// TIA Portal project "Assembler" (V15)
// Vorlageprojekt für das Buch mit Zielsystem S7-1200

(* hardware
DEVICE "S7-1200-Station_1"  S7-1200 Station
   slot 0: "Baugruppenträger_0"  Rack  V1.0
   slot 1: "PLC_1"  CPU 1211C DC/DC/DC  6ES7 211-1AE40-0XB0  V4.1
*)

// ===== PLC "PLC_1"  CPU 1211C DC/DC/DC =====

VAR_GLOBAL   // PLC tag table "Standard-Variablentabelle"
   "Clock_Byte" AT %MB0 : Byte;
   "Clock_10Hz" AT %M0.0 : Bool;
   "Clock_5Hz" AT %M0.1 : Bool;
   "Clock_2.5Hz" AT %M0.2 : Bool;
   "Clock_2Hz" AT %M0.3 : Bool;
   "Clock_1.25Hz" AT %M0.4 : Bool;
   "Clock_1Hz" AT %M0.5 : Bool;
   "Clock_0.625Hz" AT %M0.6 : Bool;
   "Clock_0.5Hz" AT %M0.7 : Bool;
END_VAR

VAR_GLOBAL   // PLC tag table "Assembler"
   "Moving X" AT %I0.0 : Bool;   // Moving X
   "Moving Z" AT %I0.1 : Bool;   // Moving Z
   "Item detected" AT %I0.2 : Bool;   // Item detected
   "Lid at place" AT %I0.3 : Bool;   // Lid at place
   "Lid clamped" AT %I0.4 : Bool;   // Lid clamped
   "Pos. at limit (lids)" AT %I0.5 : Bool;   // Pos. at limit (lids) (NC)
   "Base at place" AT %I0.6 : Bool;   // Base at place
   "Base clamped" AT %I0.7 : Bool;   // Base clamped
   "Pos. at limit (bases)" AT %I1.0 : Bool;   // Pos. at limit (bases) (NC)
   "Part leaving" AT %I1.1 : Bool;   // Part leaving
   "Start" AT %I1.2 : Bool;   // Start
   "Reset" AT %I1.3 : Bool;   // Reset
   "Stop" AT %I1.4 : Bool;   // Stop (NC)
   "Emergency stop" AT %I1.5 : Bool;   // Emergency stop (NC)
   "Auto" AT %I1.6 : Bool;   // Auto
   "FACTORY I/O (Running)" AT %I1.7 : Bool;   // FACTORY I/O (Running)
   "Move X" AT %Q0.0 : Bool;   // Move X
   "Move Z" AT %Q0.1 : Bool;   // Move Z
   "Grab" AT %Q0.2 : Bool;   // Grab
   "Lids conveyor" AT %Q0.3 : Bool;   // Lids conveyor
   "Clamp lid" AT %Q0.4 : Bool;   // Clamp lid
   "Pos. raise (lids)" AT %Q0.5 : Bool;   // Pos. raise (lids)
   "Bases conveyor" AT %Q0.6 : Bool;   // Bases conveyor
   "Clamp base" AT %Q0.7 : Bool;   // Clamp base
   "Pos. raise (bases)" AT %Q1.0 : Bool;   // Pos. raise (bases)
   "Start light" AT %Q1.1 : Bool;   // Start light
   "Reset light" AT %Q1.2 : Bool;   // Reset light
   "Stop light" AT %Q1.3 : Bool;   // Stop light
   "Counter" AT %QW30 : Int;   // Counter
END_VAR

VAR_GLOBAL   // PLC tag table "GRAFCET"
   "memReset" AT %M2.0 : Bool;   // memReset
   "memStepsOff" AT %M2.1 : Bool;   // memStepsOff
   "memInit" AT %M2.2 : Bool;   // memInit
   "Step 1" AT %M2.3 : Bool;   // Step 1
   "Step 2" AT %M2.4 : Bool;   // Step 2
   "Step 3" AT %M2.5 : Bool;   // Step 3
   "Step 4" AT %M2.6 : Bool;   // Step 4
   "Step 5" AT %M2.7 : Bool;   // Step 5
   "Step 6" AT %M3.0 : Bool;   // Step 6
   "Step 7" AT %M3.1 : Bool;   // Step 7
   "Step 8" AT %M3.2 : Bool;   // Step 8
   "Step 9" AT %M3.3 : Bool;   // Step 9
   "Step 10" AT %M3.4 : Bool;   // Step 10
   "Step 11" AT %M3.5 : Bool;   // Step 11
   "Step 12" AT %M3.6 : Bool;   // Step 12
   "Step 13" AT %M3.7 : Bool;   // Step 13
   "Step 14" AT %M4.0 : Bool;   // Step 14
   "Step 15" AT %M4.1 : Bool;   // Step 15
   "N Lid at place" AT %M4.2 : Bool;   // Neg edge for Lid at place
   "N Base at place" AT %M4.3 : Bool;   // Neg edge for Base at place
   "N Moving Z1" AT %M4.4 : Bool;   // Neg edge for Moving Z1
   "N Moving X" AT %M4.6 : Bool;   // Neg edge for Moving X
   "N Part leaving" AT %M4.7 : Bool;   // Neg edge for Part leaving
   "N Moving Z2" AT %M4.5 : Bool;   // Neg edge for Moving Z2
   "Auto Flag" AT %M5.0 : Bool;   // Auto Flag
   "Manual Flag" AT %M5.1 : Bool;   // Manual Flag
END_VAR

// folder: System blocks/Program resources

DATA_BLOCK "Parts Counter"   // DB1
{ S7_Optimized_Access := 'TRUE' }
AUTHOR : Simatic
FAMILY : IEC
NAME : CNTR
VERSION : 1.0
// stored: InstanceOfName IEC_COUNTER
"IEC_COUNTER"
BEGIN
END_DATA_BLOCK

// folder: (top level)

FUNCTION "Steps" : Void   // FC1, LAD
{ S7_Optimized_Access := 'TRUE' }
VERSION : 0.1
   VAR_TEMP   // added for the SCL form of the ladder/FBD networks
      _w1 : Bool;
   END_VAR
BEGIN

REGION Network 1: Manual Flag
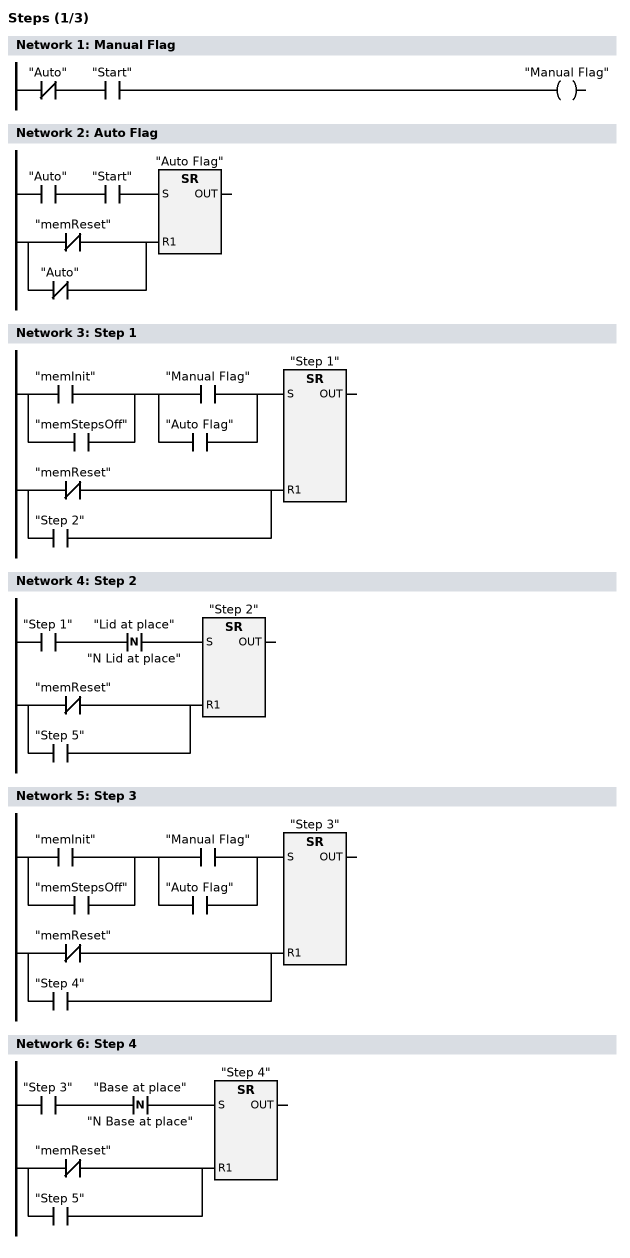
   RUNG wire#powerrail
      I_Contact( "Auto" )
      Contact( "Start" )
      Coil( "Manual Flag" )
   END_RUNG
   // the same network as SCL:
   "Manual Flag" := NOT "Auto" AND "Start";
END_REGION

REGION Network 2: Auto Flag
   RUNG wire#powerrail
      Contact( "Auto" )
      Contact( "Start" )
      S_SR(operand := "Auto Flag", r1 := wire#w1)
   END_RUNG
   RUNG wire#powerrail
      I_Contact( "memReset" )
   END_RUNG wire#w1
   RUNG wire#powerrail
      I_Contact( "Auto" )
   END_RUNG wire#w1
   // the same network as SCL:
   IF "Auto" AND "Start" THEN
       "Auto Flag" := TRUE;   // SR flip-flop
   END_IF;
   IF NOT "memReset" OR NOT "Auto" THEN "Auto Flag" := FALSE; END_IF;
END_REGION

REGION Network 3: Step 1
   RUNG wire#powerrail
      Contact( "memInit" )
      wire#w1
      Contact( "Manual Flag" )
      wire#w2
      S_SR(operand := "Step 1", r1 := wire#w3)
   END_RUNG
   RUNG wire#powerrail
      Contact( "memStepsOff" )
   END_RUNG wire#w1
   RUNG wire#w1
      Contact( "Auto Flag" )
   END_RUNG wire#w2
   RUNG wire#powerrail
      I_Contact( "memReset" )
   END_RUNG wire#w3
   RUNG wire#powerrail
      Contact( "Step 2" )
   END_RUNG wire#w3
   // the same network as SCL:
   IF ("memInit" OR "memStepsOff") AND ("Manual Flag" OR "Auto Flag") THEN
       "Step 1" := TRUE;   // SR flip-flop
   END_IF;
   IF NOT "memReset" OR "Step 2" THEN "Step 1" := FALSE; END_IF;
END_REGION

REGION Network 4: Step 2
   RUNG wire#powerrail
      Contact( "Step 1" )
      N_Contact(operand := "Lid at place", bit := "N Lid at place")
      S_SR(operand := "Step 2", r1 := wire#w1)
   END_RUNG
   RUNG wire#powerrail
      I_Contact( "memReset" )
   END_RUNG wire#w1
   RUNG wire#powerrail
      Contact( "Step 5" )
   END_RUNG wire#w1
   // the same network as SCL:
   #_w1 := "Step 1" AND NOT "Lid at place" AND "N Lid at place";   // falling edge of "Lid at place"
   "N Lid at place" := "Lid at place";
   IF #_w1 THEN
       "Step 2" := TRUE;   // SR flip-flop
   END_IF;
   IF NOT "memReset" OR "Step 5" THEN "Step 2" := FALSE; END_IF;
END_REGION

REGION Network 5: Step 3
   RUNG wire#powerrail
      Contact( "memInit" )
      wire#w1
      Contact( "Manual Flag" )
      wire#w2
      S_SR(operand := "Step 3", r1 := wire#w3)
   END_RUNG
   RUNG wire#powerrail
      Contact( "memStepsOff" )
   END_RUNG wire#w1
   RUNG wire#w1
      Contact( "Auto Flag" )
   END_RUNG wire#w2
   RUNG wire#powerrail
      I_Contact( "memReset" )
   END_RUNG wire#w3
   RUNG wire#powerrail
      Contact( "Step 4" )
   END_RUNG wire#w3
   // the same network as SCL:
   IF ("memInit" OR "memStepsOff") AND ("Manual Flag" OR "Auto Flag") THEN
       "Step 3" := TRUE;   // SR flip-flop
   END_IF;
   IF NOT "memReset" OR "Step 4" THEN "Step 3" := FALSE; END_IF;
END_REGION

REGION Network 6: Step 4
   RUNG wire#powerrail
      Contact( "Step 3" )
      N_Contact(operand := "Base at place", bit := "N Base at place")
      S_SR(operand := "Step 4", r1 := wire#w1)
   END_RUNG
   RUNG wire#powerrail
      I_Contact( "memReset" )
   END_RUNG wire#w1
   RUNG wire#powerrail
      Contact( "Step 5" )
   END_RUNG wire#w1
   // the same network as SCL:
   #_w1 := "Step 3" AND NOT "Base at place" AND "N Base at place";   // falling edge of "Base at place"
   "N Base at place" := "Base at place";
   IF #_w1 THEN
       "Step 4" := TRUE;   // SR flip-flop
   END_IF;
   IF NOT "memReset" OR "Step 5" THEN "Step 4" := FALSE; END_IF;
END_REGION

REGION Network 7: Step 5
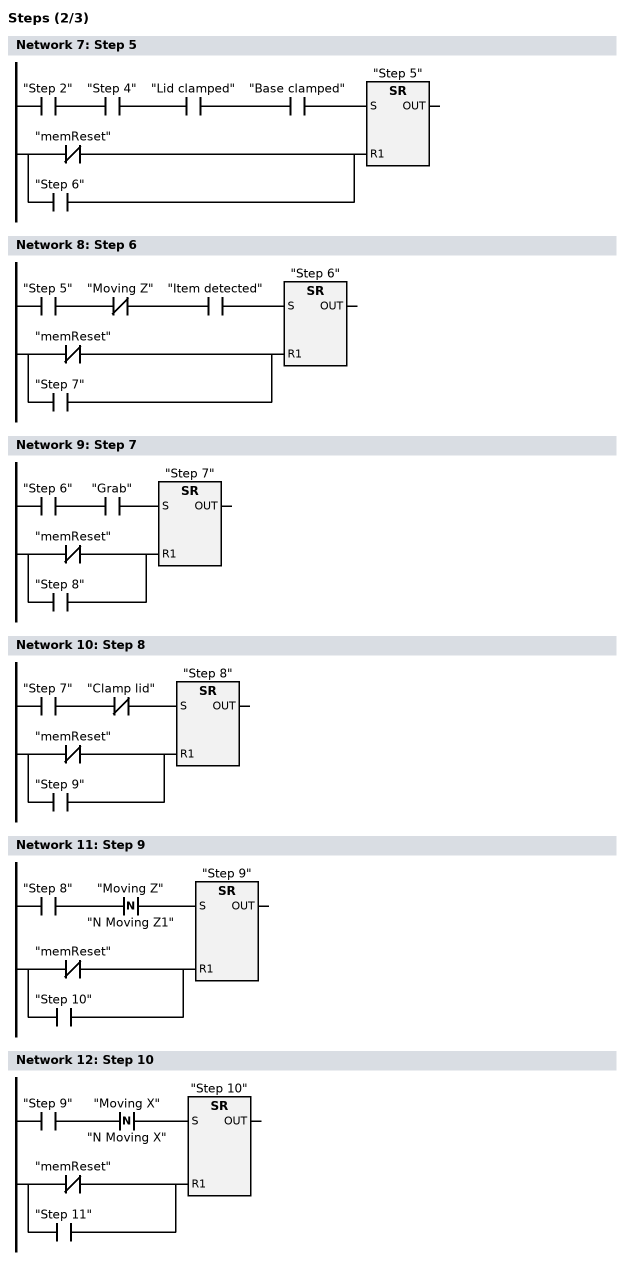
   RUNG wire#powerrail
      Contact( "Step 2" )
      Contact( "Step 4" )
      Contact( "Lid clamped" )
      Contact( "Base clamped" )
      S_SR(operand := "Step 5", r1 := wire#w1)
   END_RUNG
   RUNG wire#powerrail
      I_Contact( "memReset" )
   END_RUNG wire#w1
   RUNG wire#powerrail
      Contact( "Step 6" )
   END_RUNG wire#w1
   // the same network as SCL:
   IF "Step 2" AND "Step 4" AND "Lid clamped" AND "Base clamped" THEN
       "Step 5" := TRUE;   // SR flip-flop
   END_IF;
   IF NOT "memReset" OR "Step 6" THEN "Step 5" := FALSE; END_IF;
END_REGION

REGION Network 8: Step 6
   RUNG wire#powerrail
      Contact( "Step 5" )
      I_Contact( "Moving Z" )
      Contact( "Item detected" )
      S_SR(operand := "Step 6", r1 := wire#w1)
   END_RUNG
   RUNG wire#powerrail
      I_Contact( "memReset" )
   END_RUNG wire#w1
   RUNG wire#powerrail
      Contact( "Step 7" )
   END_RUNG wire#w1
   // the same network as SCL:
   IF "Step 5" AND NOT "Moving Z" AND "Item detected" THEN
       "Step 6" := TRUE;   // SR flip-flop
   END_IF;
   IF NOT "memReset" OR "Step 7" THEN "Step 6" := FALSE; END_IF;
END_REGION

REGION Network 9: Step 7
   RUNG wire#powerrail
      Contact( "Step 6" )
      Contact( "Grab" )
      S_SR(operand := "Step 7", r1 := wire#w1)
   END_RUNG
   RUNG wire#powerrail
      I_Contact( "memReset" )
   END_RUNG wire#w1
   RUNG wire#powerrail
      Contact( "Step 8" )
   END_RUNG wire#w1
   // the same network as SCL:
   IF "Step 6" AND "Grab" THEN
       "Step 7" := TRUE;   // SR flip-flop
   END_IF;
   IF NOT "memReset" OR "Step 8" THEN "Step 7" := FALSE; END_IF;
END_REGION

REGION Network 10: Step 8
   RUNG wire#powerrail
      Contact( "Step 7" )
      I_Contact( "Clamp lid" )
      S_SR(operand := "Step 8", r1 := wire#w1)
   END_RUNG
   RUNG wire#powerrail
      I_Contact( "memReset" )
   END_RUNG wire#w1
   RUNG wire#powerrail
      Contact( "Step 9" )
   END_RUNG wire#w1
   // the same network as SCL:
   IF "Step 7" AND NOT "Clamp lid" THEN
       "Step 8" := TRUE;   // SR flip-flop
   END_IF;
   IF NOT "memReset" OR "Step 9" THEN "Step 8" := FALSE; END_IF;
END_REGION

REGION Network 11: Step 9
   RUNG wire#powerrail
      Contact( "Step 8" )
      N_Contact(operand := "Moving Z", bit := "N Moving Z1")
      S_SR(operand := "Step 9", r1 := wire#w1)
   END_RUNG
   RUNG wire#powerrail
      I_Contact( "memReset" )
   END_RUNG wire#w1
   RUNG wire#powerrail
      Contact( "Step 10" )
   END_RUNG wire#w1
   // the same network as SCL:
   #_w1 := "Step 8" AND NOT "Moving Z" AND "N Moving Z1";   // falling edge of "Moving Z"
   "N Moving Z1" := "Moving Z";
   IF #_w1 THEN
       "Step 9" := TRUE;   // SR flip-flop
   END_IF;
   IF NOT "memReset" OR "Step 10" THEN "Step 9" := FALSE; END_IF;
END_REGION

REGION Network 12: Step 10
   RUNG wire#powerrail
      Contact( "Step 9" )
      N_Contact(operand := "Moving X", bit := "N Moving X")
      S_SR(operand := "Step 10", r1 := wire#w1)
   END_RUNG
   RUNG wire#powerrail
      I_Contact( "memReset" )
   END_RUNG wire#w1
   RUNG wire#powerrail
      Contact( "Step 11" )
   END_RUNG wire#w1
   // the same network as SCL:
   #_w1 := "Step 9" AND NOT "Moving X" AND "N Moving X";   // falling edge of "Moving X"
   "N Moving X" := "Moving X";
   IF #_w1 THEN
       "Step 10" := TRUE;   // SR flip-flop
   END_IF;
   IF NOT "memReset" OR "Step 11" THEN "Step 10" := FALSE; END_IF;
END_REGION

REGION Network 13: Step 11
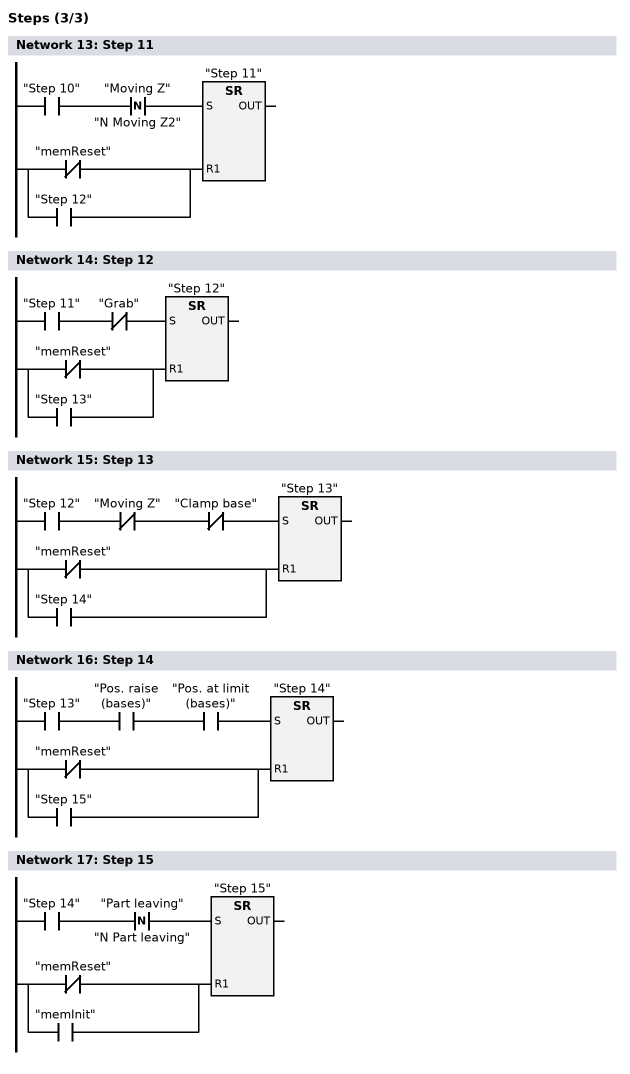
   RUNG wire#powerrail
      Contact( "Step 10" )
      N_Contact(operand := "Moving Z", bit := "N Moving Z2")
      S_SR(operand := "Step 11", r1 := wire#w1)
   END_RUNG
   RUNG wire#powerrail
      I_Contact( "memReset" )
   END_RUNG wire#w1
   RUNG wire#powerrail
      Contact( "Step 12" )
   END_RUNG wire#w1
   // the same network as SCL:
   #_w1 := "Step 10" AND NOT "Moving Z" AND "N Moving Z2";   // falling edge of "Moving Z"
   "N Moving Z2" := "Moving Z";
   IF #_w1 THEN
       "Step 11" := TRUE;   // SR flip-flop
   END_IF;
   IF NOT "memReset" OR "Step 12" THEN "Step 11" := FALSE; END_IF;
END_REGION

REGION Network 14: Step 12
   RUNG wire#powerrail
      Contact( "Step 11" )
      I_Contact( "Grab" )
      S_SR(operand := "Step 12", r1 := wire#w1)
   END_RUNG
   RUNG wire#powerrail
      I_Contact( "memReset" )
   END_RUNG wire#w1
   RUNG wire#powerrail
      Contact( "Step 13" )
   END_RUNG wire#w1
   // the same network as SCL:
   IF "Step 11" AND NOT "Grab" THEN
       "Step 12" := TRUE;   // SR flip-flop
   END_IF;
   IF NOT "memReset" OR "Step 13" THEN "Step 12" := FALSE; END_IF;
END_REGION

REGION Network 15: Step 13
   RUNG wire#powerrail
      Contact( "Step 12" )
      I_Contact( "Moving Z" )
      I_Contact( "Clamp base" )
      S_SR(operand := "Step 13", r1 := wire#w1)
   END_RUNG
   RUNG wire#powerrail
      I_Contact( "memReset" )
   END_RUNG wire#w1
   RUNG wire#powerrail
      Contact( "Step 14" )
   END_RUNG wire#w1
   // the same network as SCL:
   IF "Step 12" AND NOT "Moving Z" AND NOT "Clamp base" THEN
       "Step 13" := TRUE;   // SR flip-flop
   END_IF;
   IF NOT "memReset" OR "Step 14" THEN "Step 13" := FALSE; END_IF;
END_REGION

REGION Network 16: Step 14
   RUNG wire#powerrail
      Contact( "Step 13" )
      Contact( "Pos. raise (bases)" )
      Contact( "Pos. at limit (bases)" )
      S_SR(operand := "Step 14", r1 := wire#w1)
   END_RUNG
   RUNG wire#powerrail
      I_Contact( "memReset" )
   END_RUNG wire#w1
   RUNG wire#powerrail
      Contact( "Step 15" )
   END_RUNG wire#w1
   // the same network as SCL:
   IF "Step 13" AND "Pos. raise (bases)" AND "Pos. at limit (bases)" THEN
       "Step 14" := TRUE;   // SR flip-flop
   END_IF;
   IF NOT "memReset" OR "Step 15" THEN "Step 14" := FALSE; END_IF;
END_REGION

REGION Network 17: Step 15
   RUNG wire#powerrail
      Contact( "Step 14" )
      N_Contact(operand := "Part leaving", bit := "N Part leaving")
      S_SR(operand := "Step 15", r1 := wire#w1)
   END_RUNG
   RUNG wire#powerrail
      I_Contact( "memReset" )
   END_RUNG wire#w1
   RUNG wire#powerrail
      Contact( "memInit" )
   END_RUNG wire#w1
   // the same network as SCL:
   #_w1 := "Step 14" AND NOT "Part leaving" AND "N Part leaving";   // falling edge of "Part leaving"
   "N Part leaving" := "Part leaving";
   IF #_w1 THEN
       "Step 15" := TRUE;   // SR flip-flop
   END_IF;
   IF NOT "memReset" OR "memInit" THEN "Step 15" := FALSE; END_IF;
END_REGION
END_FUNCTION

FUNCTION "Actions" : Void   // FC2, LAD
{ S7_Optimized_Access := 'TRUE' }
VERSION : 0.1
BEGIN

REGION Network 1: Lids conveyor
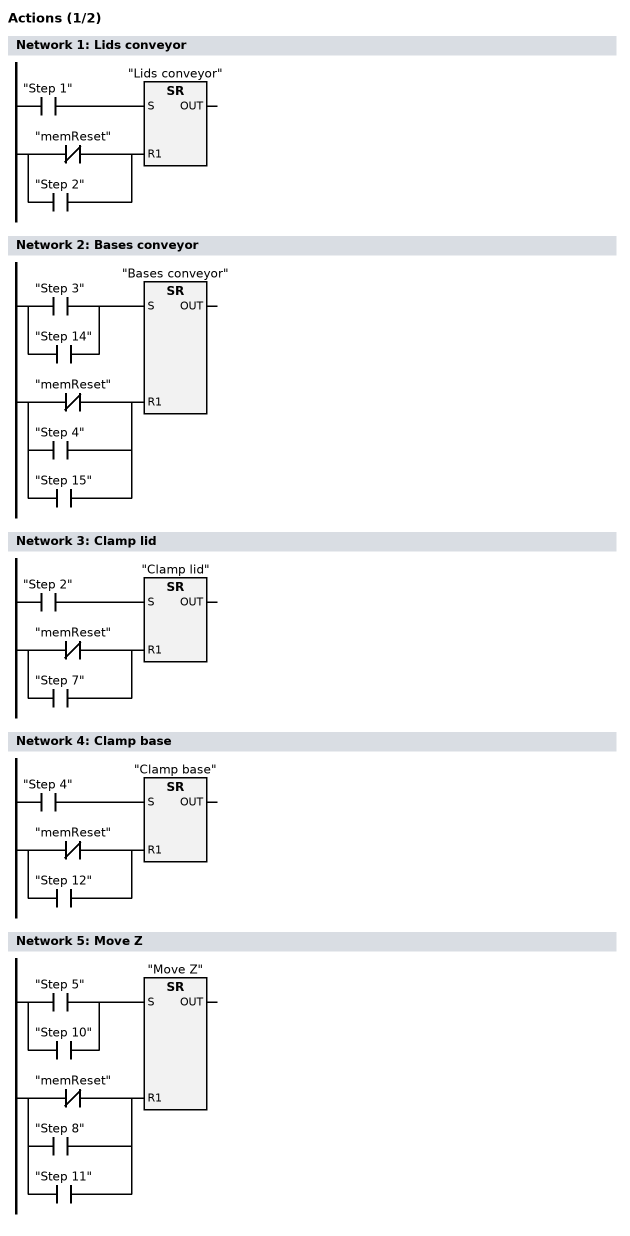
   RUNG wire#powerrail
      Contact( "Step 1" )
      S_SR(operand := "Lids conveyor", r1 := wire#w1)
   END_RUNG
   RUNG wire#powerrail
      I_Contact( "memReset" )
   END_RUNG wire#w1
   RUNG wire#powerrail
      Contact( "Step 2" )
   END_RUNG wire#w1
   // the same network as SCL:
   IF "Step 1" THEN
       "Lids conveyor" := TRUE;   // SR flip-flop
   END_IF;
   IF NOT "memReset" OR "Step 2" THEN "Lids conveyor" := FALSE; END_IF;
END_REGION

REGION Network 2: Bases conveyor
   RUNG wire#powerrail
      Contact( "Step 3" )
      wire#w1
      S_SR(operand := "Bases conveyor", r1 := wire#w2)
   END_RUNG
   RUNG wire#powerrail
      Contact( "Step 14" )
   END_RUNG wire#w1
   RUNG wire#powerrail
      I_Contact( "memReset" )
   END_RUNG wire#w2
   RUNG wire#powerrail
      Contact( "Step 4" )
   END_RUNG wire#w2
   RUNG wire#powerrail
      Contact( "Step 15" )
   END_RUNG wire#w2
   // the same network as SCL:
   IF "Step 3" OR "Step 14" THEN
       "Bases conveyor" := TRUE;   // SR flip-flop
   END_IF;
   IF NOT "memReset" OR "Step 4" OR "Step 15" THEN "Bases conveyor" := FALSE; END_IF;
END_REGION

REGION Network 3: Clamp lid
   RUNG wire#powerrail
      Contact( "Step 2" )
      S_SR(operand := "Clamp lid", r1 := wire#w1)
   END_RUNG
   RUNG wire#powerrail
      I_Contact( "memReset" )
   END_RUNG wire#w1
   RUNG wire#powerrail
      Contact( "Step 7" )
   END_RUNG wire#w1
   // the same network as SCL:
   IF "Step 2" THEN
       "Clamp lid" := TRUE;   // SR flip-flop
   END_IF;
   IF NOT "memReset" OR "Step 7" THEN "Clamp lid" := FALSE; END_IF;
END_REGION

REGION Network 4: Clamp base
   RUNG wire#powerrail
      Contact( "Step 4" )
      S_SR(operand := "Clamp base", r1 := wire#w1)
   END_RUNG
   RUNG wire#powerrail
      I_Contact( "memReset" )
   END_RUNG wire#w1
   RUNG wire#powerrail
      Contact( "Step 12" )
   END_RUNG wire#w1
   // the same network as SCL:
   IF "Step 4" THEN
       "Clamp base" := TRUE;   // SR flip-flop
   END_IF;
   IF NOT "memReset" OR "Step 12" THEN "Clamp base" := FALSE; END_IF;
END_REGION

REGION Network 5: Move Z
   RUNG wire#powerrail
      Contact( "Step 5" )
      wire#w1
      S_SR(operand := "Move Z", r1 := wire#w2)
   END_RUNG
   RUNG wire#powerrail
      Contact( "Step 10" )
   END_RUNG wire#w1
   RUNG wire#powerrail
      I_Contact( "memReset" )
   END_RUNG wire#w2
   RUNG wire#powerrail
      Contact( "Step 8" )
   END_RUNG wire#w2
   RUNG wire#powerrail
      Contact( "Step 11" )
   END_RUNG wire#w2
   // the same network as SCL:
   IF "Step 5" OR "Step 10" THEN
       "Move Z" := TRUE;   // SR flip-flop
   END_IF;
   IF NOT "memReset" OR "Step 8" OR "Step 11" THEN "Move Z" := FALSE; END_IF;
END_REGION

REGION Network 6: Move X
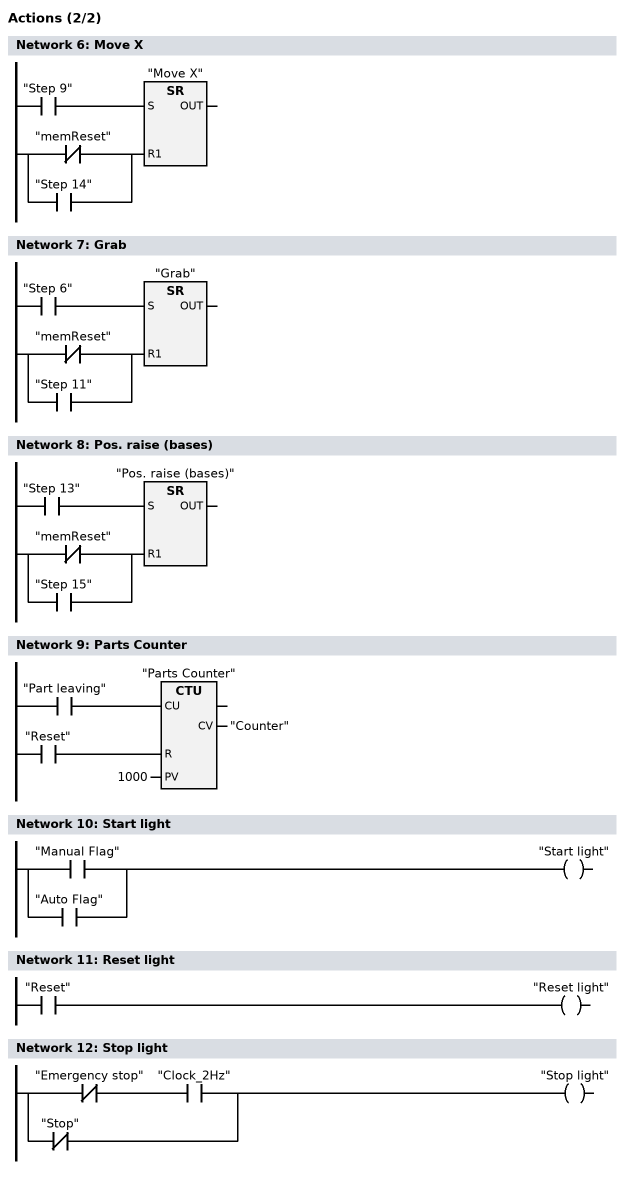
   RUNG wire#powerrail
      Contact( "Step 9" )
      S_SR(operand := "Move X", r1 := wire#w1)
   END_RUNG
   RUNG wire#powerrail
      I_Contact( "memReset" )
   END_RUNG wire#w1
   RUNG wire#powerrail
      Contact( "Step 14" )
   END_RUNG wire#w1
   // the same network as SCL:
   IF "Step 9" THEN
       "Move X" := TRUE;   // SR flip-flop
   END_IF;
   IF NOT "memReset" OR "Step 14" THEN "Move X" := FALSE; END_IF;
END_REGION

REGION Network 7: Grab
   RUNG wire#powerrail
      Contact( "Step 6" )
      S_SR(operand := "Grab", r1 := wire#w1)
   END_RUNG
   RUNG wire#powerrail
      I_Contact( "memReset" )
   END_RUNG wire#w1
   RUNG wire#powerrail
      Contact( "Step 11" )
   END_RUNG wire#w1
   // the same network as SCL:
   IF "Step 6" THEN
       "Grab" := TRUE;   // SR flip-flop
   END_IF;
   IF NOT "memReset" OR "Step 11" THEN "Grab" := FALSE; END_IF;
END_REGION

REGION Network 8: Pos. raise (bases)
   RUNG wire#powerrail
      Contact( "Step 13" )
      S_SR(operand := "Pos. raise (bases)", r1 := wire#w1)
   END_RUNG
   RUNG wire#powerrail
      I_Contact( "memReset" )
   END_RUNG wire#w1
   RUNG wire#powerrail
      Contact( "Step 15" )
   END_RUNG wire#w1
   // the same network as SCL:
   IF "Step 13" THEN
       "Pos. raise (bases)" := TRUE;   // SR flip-flop
   END_IF;
   IF NOT "memReset" OR "Step 15" THEN "Pos. raise (bases)" := FALSE; END_IF;
END_REGION

REGION Network 9: Parts Counter
   "Parts Counter".CTU(CU := "Part leaving", R := "Reset", PV := 1000, CV => "Counter");
END_REGION

REGION Network 10: Start light
   RUNG wire#powerrail
      Contact( "Manual Flag" )
      wire#w1
      Coil( "Start light" )
   END_RUNG
   RUNG wire#powerrail
      Contact( "Auto Flag" )
   END_RUNG wire#w1
   // the same network as SCL:
   "Start light" := "Manual Flag" OR "Auto Flag";
END_REGION

REGION Network 11: Reset light
   RUNG wire#powerrail
      Contact( "Reset" )
      Coil( "Reset light" )
   END_RUNG
   // the same network as SCL:
   "Reset light" := "Reset";
END_REGION

REGION Network 12: Stop light
   RUNG wire#powerrail
      I_Contact( "Emergency stop" )
      Contact( "Clock_2Hz" )
      wire#w1
      Coil( "Stop light" )
   END_RUNG
   RUNG wire#powerrail
      I_Contact( "Stop" )
   END_RUNG wire#w1
   // the same network as SCL:
   "Stop light" := (NOT "Emergency stop" AND "Clock_2Hz") OR NOT "Stop";
END_REGION
END_FUNCTION

FUNCTION "MHJ-PLC-Lab-Function-S71200" : Void   // FC9000, SCL
{ S7_Optimized_Access := 'TRUE' }
VERSION : 0.1
   VAR_TEMP
      rdTimeReturn : Int;
      outputTime : DTL;
      SyncVal : Byte;
      forVal : Int;
      forVal_2 : Int;
      Value : Byte;
   END_VAR
   VAR CONSTANT
      CompVal : Byte := 16#34;
      Value_01 : Byte := 16#11;
      Value_01_DW : DWord := 16#A165_D992;
      Value_02_DW : DWord := 16#58BE_4401;
   END_VAR
BEGIN

   #Value:=PEEK(area := 16#82,
        dbNumber := 0,
        byteOffset := 511);
   #Value := #Value + 1;

   POKE(area := 16#82,
        dbNumber := 0,
        byteOffset := 511,
        value := #Value);

   POKE(area:=16#81,
        dbNumber:=0,
        byteOffset:=1016,
        value:=#Value_01_DW);
   POKE(area := 16#81,
        dbNumber := 0,
        byteOffset := 1020,
        value := #Value_02_DW);

   POKE(area := 16#81,
        dbNumber := 0,
        byteOffset := 511,
        value := B#16#00);

   FOR #forVal := 0 TO 120 DO
       FOR #forVal_2:=0 TO 10 DO
           #rdTimeReturn:=RD_SYS_T(#outputTime);
           #rdTimeReturn := WR_SYS_T(#outputTime);
           #rdTimeReturn := RD_SYS_T(#outputTime);
           #rdTimeReturn := WR_SYS_T(#outputTime);
       END_FOR;
       #SyncVal:= PEEK(area := 16#81,
                      dbNumber := 0,
                      byteOffset := 511);
       IF #SyncVal = #CompVal THEN
          GOTO M_1;
       END_IF;
   END_FOR;
   RETURN;

   M_1:
   POKE(area := 16#81,
        dbNumber := 0,
        byteOffset := 511,
        value := B#16#0);
END_FUNCTION

ORGANIZATION_BLOCK "Main"   // OB1, LAD, ProgramCycle
TITLE = "Main Program Sweep (Cycle)"
{ S7_Optimized_Access := 'TRUE' }
VERSION : 0.1
   VAR_INPUT
      Initial_Call : Bool;   // Initial call of this OB
      Remanence : Bool;   // =True, if remanent data are available
   END_VAR
BEGIN

REGION Network 1: Konnektierungsbaustein für PLC-Lab / Factory IO Template
   // Im Netzwerk 1 wird der Konnektierungsbaustein für PLC-Lab aufgerufen.
   // Dieser Aufruf darf nicht entfernt werden!
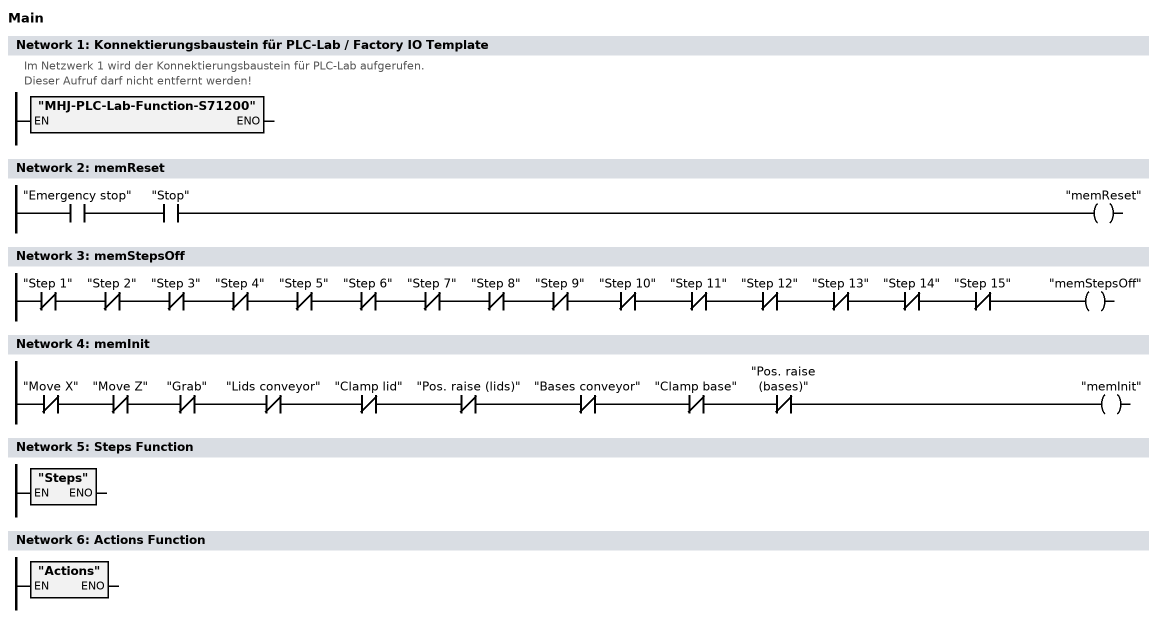
   RUNG wire#powerrail
      "MHJ-PLC-Lab-Function-S71200"()
   END_RUNG
   // the same network as SCL:
   "MHJ-PLC-Lab-Function-S71200"();
END_REGION

REGION Network 2: memReset
   RUNG wire#powerrail
      Contact( "Emergency stop" )
      Contact( "Stop" )
      Coil( "memReset" )
   END_RUNG
   // the same network as SCL:
   "memReset" := "Emergency stop" AND "Stop";
END_REGION

REGION Network 3: memStepsOff
   RUNG wire#powerrail
      I_Contact( "Step 1" )
      I_Contact( "Step 2" )
      I_Contact( "Step 3" )
      I_Contact( "Step 4" )
      I_Contact( "Step 5" )
      I_Contact( "Step 6" )
      I_Contact( "Step 7" )
      I_Contact( "Step 8" )
      I_Contact( "Step 9" )
      I_Contact( "Step 10" )
      I_Contact( "Step 11" )
      I_Contact( "Step 12" )
      I_Contact( "Step 13" )
      I_Contact( "Step 14" )
      I_Contact( "Step 15" )
      Coil( "memStepsOff" )
   END_RUNG
   // the same network as SCL:
   "memStepsOff" := NOT "Step 1" AND NOT "Step 2" AND NOT "Step 3" AND NOT "Step 4" AND NOT "Step 5" AND NOT "Step 6" AND NOT "Step 7" AND NOT "Step 8" AND NOT "Step 9" AND NOT "Step 10" AND NOT "Step 11" AND NOT "Step 12" AND NOT "Step 13" AND NOT "Step 14" AND NOT "Step 15";
END_REGION

REGION Network 4: memInit
   RUNG wire#powerrail
      I_Contact( "Move X" )
      I_Contact( "Move Z" )
      I_Contact( "Grab" )
      I_Contact( "Lids conveyor" )
      I_Contact( "Clamp lid" )
      I_Contact( "Pos. raise (lids)" )
      I_Contact( "Bases conveyor" )
      I_Contact( "Clamp base" )
      I_Contact( "Pos. raise (bases)" )
      Coil( "memInit" )
   END_RUNG
   // the same network as SCL:
   "memInit" := NOT "Move X" AND NOT "Move Z" AND NOT "Grab" AND NOT "Lids conveyor" AND NOT "Clamp lid" AND NOT "Pos. raise (lids)" AND NOT "Bases conveyor" AND NOT "Clamp base" AND NOT "Pos. raise (bases)";
END_REGION

REGION Network 5: Steps Function
   RUNG wire#powerrail
      "Steps"()
   END_RUNG
   // the same network as SCL:
   "Steps"();
END_REGION

REGION Network 6: Actions Function
   RUNG wire#powerrail
      "Actions"()
   END_RUNG
   // the same network as SCL:
   "Actions"();
END_REGION
END_ORGANIZATION_BLOCK